// TIA Portal V20 export
DATA_BLOCK "DI2"   // DB290
// stored: MemoryReserve 100
   VAR
      SPARE1 : Bool;
      "CONTROL POWER SMPS DC OK E6104PWS" : Bool;
      "ET200MP I/O OUTPUT POWER TRIPPED E6154CB" : Bool;
      "JUNCTION BOX CONTROL POWER TRIPPED E6180CB" : Bool;
      "CLASS 2 SMPS POWER TRIPPED E6204CB" : Bool;
      "CLASS 2 SMPS MONITORING E6206PWS" : Bool;
      "ET200ECO PN-1 POWER TRIPPED E6220CB" : Bool;
      "ET200ECO PN-2 POWER TRIPPED E6224CB" : Bool;
      "ET200ECO PN-3 POWER TRIPPED E6228CB" : Bool;
      SPARE2 : Bool;
      "PANEL FAN POWER TRIPPED E6304CB" : Bool;
      SPARE3 : Bool;
      "CONTROLLER POWER SMPS DC OK E6404PWS" : Bool;
      "CONTROLLER DC POWER TRIPPED E6406CB" : Bool;
      "SERVO CONTROL POWER TRIPPED E6416CB" : Bool;
      "MANIFOLD-1 CONTROL POWER TRIPPED E6422CB" : Bool;
      SPARE4 : Bool;
      "RFID POWER TRIPPED E6456CB" : Bool;
      "QR READER POWER TRIPPED E6462CB" : Bool;
      "QR READER POWER TRIPPED E6468CB" : Bool;
      SPARE5 : Bool;
      SPARE6 : Bool;
      "CONTROLLER POWER SMPS DC OK E6704PWS" : Bool;
      "CONTROLLER DC POWER TRIPPED E6706CB" : Bool;
      "HANDY QR READER POWER TRIPPED E6716CB" : Bool;
      "VISION CONTROLLER POWER TRIPPED E6722CB" : Bool;
      "LINE LASER MODULE-1 POWER TRIPPED E6728CB" : Bool;
      "LINE LASER MODULE-2 POWER TRIPPED E6734CB" : Bool;
      "EPC CONTROLLER-1 POWER TRIPPED E6756CB" : Bool;
      "EPC CONTROLLER-2 POWER TRIPPED E6762CB" : Bool;
      "EPC CONTROLLER-3 POWER TRIPPED E6768CB" : Bool;
      "DRIVE-CLIQ HUB POWER TRIPPED E6774CB" : Bool;
   END_VAR
BEGIN
END_DATA_BLOCK
